TYPE ST_Trackpad :
STRUCT
	ID: USINT;
	Active: BOOL;
	X: UINT;
	Y: UINT;
END_STRUCT
END_TYPE

(* stored: Version 1.1.0.1
   DUT ST_Trackpad: Id {d80eab9f-545b-4809-8bfc-c7c96718771a} *)
